Staubli VAL3: page_viewInstr.dtx

num nIndex
num nKey
public num nPage
num nRefresh
num nSelected
num nTime = 1
num nView
string sEvent
public string sItems
string sList
string sMenu[8]
string sMessage
string sProgram
string sMenu8[8]
bool bButton[8]
  [0] = true
  [2] = true
  [3] = true
  [4] = true
  [5] = true
  [6] = true
  [7] = true
bool bLarge
